// TIA Portal V19 export
FUNCTION "Peripherie" : Void   // FC1090, LAD
TITLE = Anlagenperipherie
{ S7_Optimized_Access := 'TRUE' }
// stored: AutoNumber false, SetENOAutomatically true
   VAR CONSTANT
      Ventilator_aus : Int := 10;
      AUS : USInt;
      Hand_EIN : USInt := 1;
      Hand_AUS : USInt := 2;
      Auto_EIN : USInt := 3;
      Auto_AUS : USInt := 4;
      STOERUNG : USInt := 5;
   END_VAR
BEGIN

REGION Network 1 (SCL): Diverses
   // Deckel Säurebecken
   "Deckel_CM01"();
   "Deckel_CM02"();
   // Schnelllauftor
   "Tor"();
END_REGION

REGION Network 2 (SCL): Sperrluftventilator
   // Frequenzumrichter [7]
   //Ansteuerung
   "Panel".Ventilator.laeuft := ("Panel".Ventilator.Auto OR "Panel".Ventilator.Ein)
   AND "DB_PNOZ_IN_Out".In.PNOZ_OK AND "DB_PNOZ_IN_Out".In.Abluft_ok AND "FU_In_Out".FU[7].PE.Statusbyte.Bereit;

   IF "Panel".Ventilator.laeuft THEN
       "A_Frg_FU_Vent" := TRUE;
   ELSIF "Panel".Ventilator.speed < #Ventilator_aus THEN
       "A_Frg_FU_Vent" := FALSE;
   END_IF;

   "FU_In_Out".FU[7].PA.Steuerwort.FrgHalt := "A_Frg_FU_Vent";
   "FU_In_Out".FU[7].PA.Steuerwort.FrgStop := "A_Frg_FU_Vent";
   "FU_In_Out".FU[7].PA.Steuerwort.RegSp := NOT "FU_In_Out".FU[7].PA.Steuerwort.FrgHalt;

   // Geschwindigkeitsvorgabe
   IF "Panel".Ventilator.laeuft THEN
       IF "Panel".Ventilator.Ein THEN
           "FU_In_Out".FU[7].PA.Speed := "Panel".Ventilator.SW_Hand * 150;
       ELSE
           IF "Uhrzeit".AZ_aktiv THEN
               "FU_In_Out".FU[7].PA.Speed := "Panel".Ventilator.SW_Auto_AZ * 150;
           ELSE
               "FU_In_Out".FU[7].PA.Speed := "Panel".Ventilator.SW_Auto_aAZ * 150;
           END_IF;
       END_IF;
   ELSE
       "FU_In_Out".FU[7].PA.Speed := 0;
   END_IF;

   // --> Panel
   "Panel".Ventilator.betriebsbereit:= "FU_In_Out".FU[7].PE.Statusbyte.Bereit;
   "Panel".Ventilator.Stoerung := "FU_In_Out".FU[7].PE.Statusbyte.Stoer;
   // SEW: 100% == 3000 U/min == 15000 Digits
   "Panel".Ventilator.speed := "FU_In_Out".FU[7].PE.Speed / 150; // in [%]

   "Status_E0A"(Hand:= "Panel".Ventilator.Ein,
                Auto:= "Panel".Ventilator.Auto,
                SonderModus_PumpeSpuelen:=FALSE,
                Stoerung:="FU_In_Out".FU[7].PE.Statusbyte.Stoer OR NOT "FU_In_Out".FU[7].PE.Statusbyte.Bereit,
                Ausgang:= "A_Frg_FU_Vent",
                StatusByte=> "Panel".Ventilator.Status);
END_REGION

REGION Network 3 (SCL): Pumpen
   // Filterpumpen Säure
   "FP_CM01.GP01"();
   "FP_CM02.GP04"();

   // Umwälzpumpen Säure
   "UP_CM01.GP02"();
   "UP_CM02.GP05"();

   // Umwälzpumpen Spüle
   "UP_CM03.GP03"();
   "UP_CM04.GP06"();

   // Versorgung GP13 / GP10
   "Pu_GP01.GP13"();
   "Pu_GP02.GP10"();

   // Entleeren Ver-/Entsorgung GP12 / GP07
   "Pu_GP01.GP12"();
   "Pu_GP02.GP07"();

   // Entleeren Pumpensümpfe GP08 / GP09
   "Pu_CL01.GP08"();
   "Pu_CL02.GP09"();

   // Pumpe GP11 Entleeren Behälter CM05
   "Pu_CM05.GP11_DB"();

   // Status Ventile
   "Ventil_Stati_DB"();
END_REGION

REGION Network 4 (SCL): Pumpe GP14 Entleeren Becken CM01..CM04
   // entsprechende Ventile / Kugelhähne müssen per Hand geöffnet werden
   // Verriegelung mit Max-Niveau Behälter CM05
   // nur Handbetrieb
   "A_CM05.GP14" := "Panel".Pu_Entleeren.Ein AND NOT "E_Niv_max_CM05.BL01";
   // Pumpe Ausschalten
   IF "E_Niv_max_CM05.BL01" THEN
       "Panel".Pu_Entleeren.Ein := FALSE;
   END_IF;
   // --> Visu
   IF "A_CM05.GP14" THEN
       "Panel".Pu_Entleeren.Status := #Hand_EIN;
   ELSE
       "Panel".Pu_Entleeren.Status := #AUS;
   END_IF;
END_REGION
END_FUNCTION
